// TwinCAT 3 PLC project MTCPLC
// ProgramVersion: 3.1.4022.3
// libraries:
//   Tc2_Standard, * (Beckhoff Automation GmbH)
//   Tc2_System, * (Beckhoff Automation GmbH)
//   Tc3_Module, * (Beckhoff Automation GmbH)
// project tree:
//   GVLs/ IO.TcGVL
//   / PlcTask.TcTTO
//   POUs/ MAIN.TcPOU, MOTOR1.TcPOU, MOTOR2.TcPOU
// real-time tasks:
//   TASK PlcTask: cycle T#10ms, priority 20, ADS port 350
// I/O:
//   DEVICE Device 1 (EtherCAT), AmsNetId 5.29.55.214.2.1
//     Term 1 (EK1100) [EK1100 EtherCAT Coupler (2A E-Bus)]
//       Term 2 (EL1008) [EL1008 8Ch. Dig. Input 24V, 3ms]
//       Term 3 (EL1008) [EL1008 8Ch. Dig. Input 24V, 3ms]
//       Term 4 (EL2008) [EL2008 8Ch. Dig. Output 24V, 0.5A]
//       Term 5 (EL2008) [EL2008 8Ch. Dig. Output 24V, 0.5A]
//       Term 6 (EL3002) [EL3002 2Ch. Ana. Input +/-10V]
//       Term 7 (EL4002) [EL4002 2Ch. Ana. Output 0-10V, 12bit]
//       Term 8 (EL3124) [EL3124 4Ch. Ana. Input 4-20mA Diff.]
//       Term 9 (EL4024) [EL4024 4Ch. Ana. Output 4-20mA, 12bit]
//       Term 10 (EL9011) [EL9011 End Terminal]
// variable links:
//   MTCPLC/MTCPLC Instance <-> Device 1 (EtherCAT)/Term 1 (EK1100)/Term 2 (EL1008)
//     PlcTask Inputs/IO.M1FaultStatus <-> Channel 4/IO.M1FaultStatus
//     PlcTask Inputs/IO.M2FaultStatus <-> Channel 6/IO.M2FaultStatus
//     PlcTask Inputs/IO.M1RunStatus <-> Channel 3/IO.M1RunStatus
//     PlcTask Inputs/IO.M2RunStatus <-> Channel 5/IO.M2RunStatus
//     PlcTask Inputs/IO.M1StartBtn <-> Channel 2/IO.M1StartBtn
//     PlcTask Inputs/IO.M1StopBtn <-> Channel 1/IO.M1StopBtn
//     PlcTask Inputs/IO.M2DirectionSwitch <-> Channel 8/IO.M2DirectionSwitch
//     PlcTask Inputs/IO.M2StartSwitch <-> Channel 7/IO.M2StartSwitch
//   MTCPLC/MTCPLC Instance <-> Device 1 (EtherCAT)/Term 1 (EK1100)/Term 3 (EL1008)
//     PlcTask Inputs/IO.M2ConstantSwitch <-> Channel 1/IO.M2ConstantSwitch
//   MTCPLC/MTCPLC Instance <-> Device 1 (EtherCAT)/Term 1 (EK1100)/Term 4 (EL2008)
//     PlcTask Outputs/IO.M1FaultLight <-> Channel 3/IO.M1FaultLight
//     PlcTask Outputs/IO.M2FaultLight <-> Channel 5/IO.M2FaultLight
//     PlcTask Outputs/IO.M1RunCommand <-> Channel 1/IO.M1RunCommand
//     PlcTask Outputs/IO.M1RunLight <-> Channel 2/IO.M1RunLight
//     PlcTask Outputs/IO.M2RunLight <-> Channel 4/IO.M2RunLight
//     PlcTask Outputs/IO.M2ConstantControl <-> Channel 8/IO.M2ConstantControl
//     PlcTask Outputs/IO.M2DirectionControl <-> Channel 7/IO.M2DirectionControl
//     PlcTask Outputs/IO.M2RunControl <-> Channel 6/IO.M2RunControl
//   MTCPLC/MTCPLC Instance <-> Device 1 (EtherCAT)/Term 1 (EK1100)/Term 6 (EL3002)
//     PlcTask Inputs/IO.AI1_1 <-> AI Standard Channel 1/IO.AI1_1
//   MTCPLC/MTCPLC Instance <-> Device 1 (EtherCAT)/Term 1 (EK1100)/Term 7 (EL4002)
//     PlcTask Outputs/IO.AQ1_1 <-> AO Outputs Channel 1/IO.AQ1_1

CONFIGURATION MTCPLC
    RESOURCE PLC ON TwinCAT3
        TASK PlcTask(INTERVAL := T#10ms, PRIORITY := 20);
        PROGRAM MAIN WITH PlcTask : MAIN;
    END_RESOURCE
END_CONFIGURATION

// ---- GVLs/IO.TcGVL
{attribute 'qualified_only'}
VAR_GLOBAL
	// DIGITAL INPUT 
	M1StopBtn AT %I* :  BOOL;
	M1StartBtn AT %I* :  BOOL;
	M1RunStatus AT %I* :  BOOL;
	M1FaultStatus AT %I* :  BOOL;
	M2RunStatus AT %I* :  BOOL;
	M2FaultStatus AT %I* :  BOOL;
	M2StartSwitch AT %I* :  BOOL;
	M2DirectionSwitch AT %I* :  BOOL;
	M2ConstantSwitch AT %I* : 	BOOL;
	
	

	// DIGITAL OUTPUT
	M1RunCommand AT %Q* : BOOL;
	M1RunLight AT %Q* : BOOL;
	M1FaultLight AT %Q* : BOOL;
	M2RunLight AT %Q* : BOOL;
	M2FaultLight AT %Q* : BOOL;
	M2RunControl AT %Q* : BOOL;
	M2DirectionControl AT %Q* : BOOL;
	M2ConstantControl AT %Q* : BOOL;
	
	// ANALOG INPUT 
	AI1_1 AT %I* : INT;
	
	// ANALOG OUTPUT 
	AQ1_1 AT %Q* : INT; 
	
END_VAR

// ---- POUs/MAIN.TcPOU
PROGRAM MAIN
VAR
END_VAR

//MTCPLC();
MOTOR1 ();
MOTOR2 ();

END_PROGRAM

// ---- POUs/MOTOR1.TcPOU
PROGRAM MOTOR1
VAR
	iStep : INT ;
	fbRising: R_TRIG;
	fbFalling: F_TRIG;
	bM1DirectionSwitch: BOOL;
	bM1RunOtherDirection: BOOL;
END_VAR

io.M1FaultLight := io.M1FaultStatus;
io.M1RunLight := io.M1RunStatus;

fbRising(CLK:= io.M1StartBtn, Q=> );
fbFalling(CLK:= (io.M1StopBtn), Q=> );

IF fbRising.Q AND io.M1StopBtn THEN 
	//IF bM1DirectionSwitch THEN
		io.M1RunCommand := TRUE;
		//bM1RunOtherDirection := FALSE;
	//ELSE
		//io.M1RunCommand := FALSE;
		//bM1RunOtherDirection := TRUE;
	//END_IF
END_IF

IF fbFalling.Q THEN 
	io.M1RunCommand := FALSE;
END_IF

END_PROGRAM

// ---- POUs/MOTOR2.TcPOU
PROGRAM MOTOR2
VAR
END_VAR

io.M2RunControl := io.M2StartSwitch;
io.M2DirectionControl := io.M2DirectionSwitch;
io.M2ConstantControl := io.M2ConstantSwitch;

io.M2RunLight := io.M2RunStatus;
io.M2FaultLight := io.M2FaultStatus;


io.AI1_1 := io.AQ1_1;

END_PROGRAM
